// TIA Portal V17 export
// export: Created 2025-03-05T07:58:58.0992941Z, ExportSetting WithDefaults, DisplayName Totally Integrated Automation Portal, DisplayVersion V17 Update 8, DisplayName TIA Portal Openness, DisplayVersion V17 Update 8, DisplayName TIA Portal Version Control Interface, DisplayVersion V17, DisplayName SINAMICS Startdrive Advanced, DisplayVersion V17 SP2, DisplayName SINAMICS Startdrive G110M, G120, G120C, G120D, G120P, G115D, DisplayVersion V17 SP2, DisplayName SINAMICS Startdrive G130, G150, S120, S150, SINAMICS MV, S210, DisplayVersion V17 SP2, DisplayName STEP 7 Professional, DisplayVersion V17 Update 8, DisplayName SINUMERIK ONE STEP 7 Toolbox, DisplayVersion V17 Update 12, DisplayName SINUMERIK 840D sl STEP 7 Toolbox, DisplayVersion V17 Update 12, DisplayName STEP 7 Safety, DisplayVersion V17 Update 6, DisplayName WinCC Advanced, DisplayVersion V17 Update 8
ORGANIZATION_BLOCK "OB121_SYNCHRONF1"   // OB121, LAD, ProgrammingError
{ S7_Optimized_Access := 'FALSE' }
VERSION : 0.0
// stored: IsIECCheckEnabled false, SetENOAutomatically false
   VAR_TEMP
      TEMP0 : Byte;
      TEMP1 : Byte;
      TEMP2 : Byte;
      TEMP3 : Byte;
      TEMP4 : Byte;
      TEMP5 : Byte;
      TEMP6 : Word;
      TEMP7 : Word;
      TEMP8 : Word;
      TEMP9 : Date_And_Time;
   END_VAR
BEGIN
END_ORGANIZATION_BLOCK
